FUNCTION_BLOCK T_ExternalControllersCollectionNotifyStateChangedSuccess EXTENDS T_UnitTestBase
VAR
  list : T_ExternalControllerCollection(10);
  newController, newController2 : T_ExternalControllerMock; 
  actual1, actual2 : BOOL;
END_VAR

// Arrange
list.AddController(newController);
list.AddController(newController2);

//Act
list.NotifyStateChanged(Tc3_PackML_V2.E_PMLCommand.ePMLCommand_Complete);

//Assert
actual1 := newController._newState = Tc3_PackML_V2.E_PMLCommand.ePMLCommand_Complete;
actual2 := newController2._newState = Tc3_PackML_V2.E_PMLCommand.ePMLCommand_Complete;

assertion.AssertEquals_BOOL(TRUE, actual1, 'newController._newState = Tc3_PackML_V2.E_PMLCommand.ePMLCommand_Complete');
assertion.AssertEquals_BOOL(TRUE, actual2, 'newController2._newState = Tc3_PackML_V2.E_PMLCommand.ePMLCommand_Complete');
TestFinished();

END_FUNCTION_BLOCK

(* stored: Version 1.1.0.1, ProductVersion 3.1.4024.12
   POU T_ExternalControllersCollectionNotifyStateChangedSuccess: Id {6096ac06-1ab7-4462-928e-01de7f658392}, SpecialFunc None *)
